(* IEC 61131-3 sources: CodesysTest/alpha/export/PackML/Pregis/PackML_Base_State_Machine_2.pou, 1 file *)

(* ---- PackML_Base_State_Machine_2.pou.st ---- *)
(*#-#-#-#-#-#-#-#-#-#---Declaration---#-#-#-#-#-#-#-#-#-#-#-#-#*)

FUNCTION_BLOCK PackML_Base_State_Machine_2
VAR_INPUT
	Reset: BOOL;
	Clear: BOOL;
	Stop: BOOL;
	Hold: BOOL;
	Suspend: BOOL;
	Abort: BOOL;
END_VAR
VAR_OUTPUT
END_VAR
VAR

	Start: BOOL;
END_VAR
